(* CODESYS project Cipher-Bay_RECOVERED_2026-03-25T10-42-59.project

Project tree, tasks and I/O mapping:
  Device : CODESYS Control for Linux SL, CODESYS, order no. 2302000005, version 4.19.0.0
    application Application
      libraries: Standard, 3.5.18.0 (System); CmpBitmapPool, * (System)
      task VISU_TASK (cyclic, interval 100 ms, priority 31) calls VisuElems.Visu_Prg
      task MainTask (cyclic, interval t#20ms, priority 1) calls PLC_PRG
      Visualization/
        visualisation VIS_Monitoring
        visualisation VIS_Home
        visualisation VIS_ControlPanel
      POUs/
        program PLC_PRG [ST]
      GLVs/
        global variables GVL_DroneDock
      DUTs/
        data type E_DockState
      External/
        image pool ImagePool
    Ethernet : Ethernet, CODESYS, version 4.2.0.0
        settings: IPAddress = [192,168,0,1]; SubnetMask = [255,255,255,0]; GatewayAddress = [0,0,0,0]; MACAddress = [16#00,16#00,16#00,16#00,16#00,16#00]; NetworkInterfaceName = 'eth0'; NetworkInterfaceName = "eth0"; SaveCommunicationSettings = FALSE; IPAddress = [192,168,0,2]; SubnetMask = [255,255,255,0]; GatewayAddress = [0,0,0,0]
      ModbusTCP_Server_Device : ModbusTCP Server Device, CODESYS, version 4.5.0.0
          settings: DistinctBitAreas = TRUE; Discrete Inputs Size = 16; StartAdresses.DiscreteInputs = 16
          output Application.GVL_DroneDock.mb_iState : WORD  // Input Registers.Input Registers
          output Application.GVL_DroneDock.mb_iBatteryLevel : WORD  // Input Registers.Input Registers
          output Application.GVL_DroneDock.mb_iChargeCurrent : WORD  // Input Registers.Input Registers
          output Application.GVL_DroneDock.xIsDocked : BOOL  // Discrete Inputs.Discrete Inputs.Bit0
          output Application.GVL_DroneDock.xIsCharging : BOOL  // Discrete Inputs.Discrete Inputs.Bit1
          unmapped channels: Holding Registers, Input Registers, Discrete Inputs
    SoftMotion General Axis Pool
  libraries: VisuSymbols, 4.5.0.0 (System); WagoVisuIcons, 1.1.0.9 (WAGO); WagoVisuIconsMaterialDesign, 1.0.0.2 (WAGO)
  text list GlobalTextList
*)

// Device/Application/DUTs/E_DockState
{attribute 'qualified_only'}
{attribute 'strict'}
TYPE E_DockState :
(
	CLOSED := 0,
    OPENING := 1,
    OPEN := 2,
    CLOSING := 3
);
END_TYPE

// Device/Application/GLVs/GVL_DroneDock
VAR_GLOBAL CONSTANT
    // Best Practice: No Magic Numbers
    MAX_BATTERY_LEVEL    : REAL := 100.0;
    CHARGE_CURRENT_MAX   : REAL := 5.2;   // Amps
    CHARGE_RATE_SIM      : REAL := 0.5;   // % added per tick for simulation
    DOOR_TRANSITION_TIME : TIME := T#4S;  // Time it takes to open/close
END_VAR

VAR_GLOBAL
    // HMI Inputs (WebVisu)
    xCmdOpen             : BOOL;
    xCmdClose            : BOOL;
    xCmdSimulateDocking  : BOOL; // Toggle to simulate drone landing

    // System Status
    eCurrentState        : E_DockState := E_DockState.CLOSED;
    xIsDocked            : BOOL;
    xIsCharging          : BOOL;
    rBatteryLevel        : REAL := 20.0; // Start at 20%
    rChargeCurrent       : REAL;

    // Modbus Variables (Scaled for 16-bit Holding Registers)
    // Modbus doesn't handle REALs natively well, so we scale REAL * 10 into INTs
    mb_iState            : WORD;  
	mb_iBatteryLevel     : WORD;  
	mb_iChargeCurrent    : WORD;
    mb_xIsDocked         : BOOL; // Coil
    mb_xIsCharging       : BOOL; // Coil
END_VAR

// Device/Application/POUs/PLC_PRG
PROGRAM PLC_PRG
VAR
	tonDoorTimer   : TON;   // Timer for door opening/closing
    tonChargePulse : TON;   // Timer to pulse the charging simulation
END_VAR

// ==========================================
// 1. DOOR CONTROL STATE MACHINE
// ==========================================
tonDoorTimer(PT := GVL_DroneDock.DOOR_TRANSITION_TIME);

CASE GVL_DroneDock.eCurrentState OF
    
    E_DockState.CLOSED:
        tonDoorTimer(IN := FALSE);
        IF GVL_DroneDock.xCmdOpen THEN
            GVL_DroneDock.xCmdOpen := FALSE; // Consume command
            GVL_DroneDock.eCurrentState := E_DockState.OPENING;
        END_IF

    E_DockState.OPENING:
        tonDoorTimer(IN := TRUE);
        IF tonDoorTimer.Q THEN
            GVL_DroneDock.eCurrentState := E_DockState.OPEN;
        END_IF
        
    E_DockState.OPEN:
        tonDoorTimer(IN := FALSE);
        IF GVL_DroneDock.xCmdClose THEN
            GVL_DroneDock.xCmdClose := FALSE; // Consume command
            GVL_DroneDock.eCurrentState := E_DockState.CLOSING;
        END_IF
        
    E_DockState.CLOSING:
        tonDoorTimer(IN := TRUE);
        IF tonDoorTimer.Q THEN
            GVL_DroneDock.eCurrentState := E_DockState.CLOSED;
        END_IF
        
END_CASE

// ==========================================
// 2. DOCKING & CHARGING SIMULATION LOGIC
// ==========================================
// Drone can only be docked/undocked if the doors are OPEN
IF GVL_DroneDock.eCurrentState = E_DockState.OPEN THEN
    GVL_DroneDock.xIsDocked := GVL_DroneDock.xCmdSimulateDocking;
END_IF

// Charging Logic: Must be docked and doors CLOSED (safe to charge)
IF GVL_DroneDock.xIsDocked AND (GVL_DroneDock.eCurrentState = E_DockState.CLOSED) THEN
    
    IF GVL_DroneDock.rBatteryLevel < GVL_DroneDock.MAX_BATTERY_LEVEL THEN
        GVL_DroneDock.xIsCharging := TRUE;
        GVL_DroneDock.rChargeCurrent := GVL_DroneDock.CHARGE_CURRENT_MAX;
        
        // Simulation: Increase battery level every 1 second
        tonChargePulse(IN := NOT tonChargePulse.Q, PT := T#1S);
        IF tonChargePulse.Q THEN
            GVL_DroneDock.rBatteryLevel := GVL_DroneDock.rBatteryLevel + GVL_DroneDock.CHARGE_RATE_SIM;
        END_IF
    ELSE
        // Battery Full
        GVL_DroneDock.xIsCharging := FALSE;
        GVL_DroneDock.rChargeCurrent := 0.0;
        GVL_DroneDock.rBatteryLevel := GVL_DroneDock.MAX_BATTERY_LEVEL;
    END_IF
    
ELSE
    // Not docked or doors open
    GVL_DroneDock.xIsCharging := FALSE;
    GVL_DroneDock.rChargeCurrent := 0.0;
    tonChargePulse(IN := FALSE);
END_IF

// ==========================================
// 3. MODBUS DATA PREPARATION
// ==========================================
// Convert Enums and REALs into standard WORDs for Modbus transmission
GVL_DroneDock.mb_iState         := INT_TO_WORD(GVL_DroneDock.eCurrentState);
GVL_DroneDock.mb_iBatteryLevel  := REAL_TO_WORD(GVL_DroneDock.rBatteryLevel * 10.0);
GVL_DroneDock.mb_iChargeCurrent := REAL_TO_WORD(GVL_DroneDock.rChargeCurrent * 10.0);
GVL_DroneDock.mb_xIsDocked      := GVL_DroneDock.xIsDocked;
GVL_DroneDock.mb_xIsCharging    := GVL_DroneDock.xIsCharging;

END_PROGRAM

// Device/Application/Visualization/VIS_Monitoring
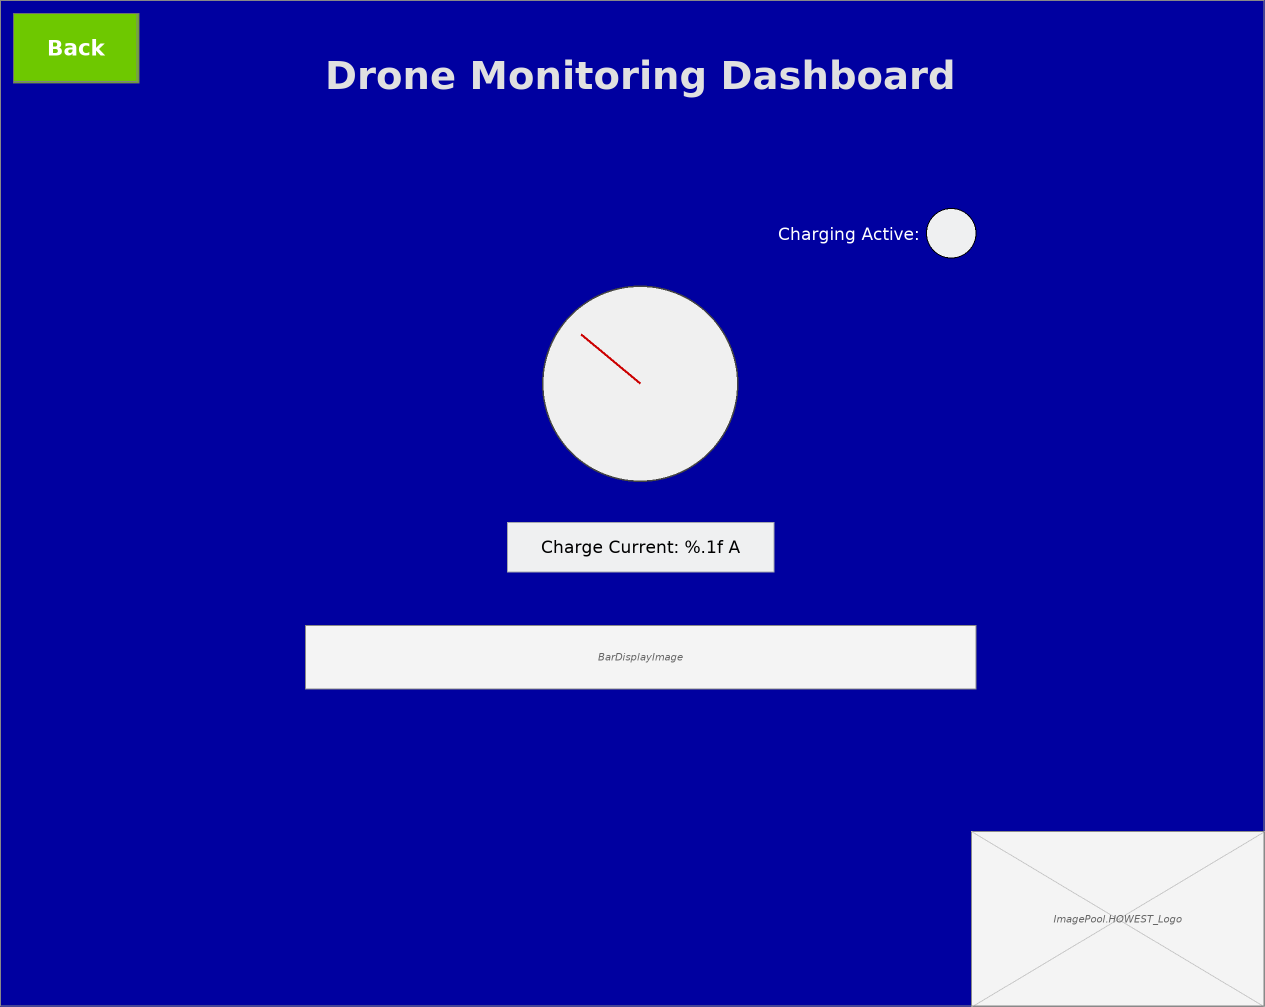
VISUALIZATION VIS_Monitoring  // 1265x1007
    Button (13,13 126x70), "Back"
        OnMouseClick:  Assign=VIS_Home, Type=Assignment
    Label (305,32 671x87), "Drone Monitoring Dashboard"
    BarDisplayImage (305,625 671x64), value: rBatteryLevel, style: BarDisplayImage-Green, scale format: %.1f, scale 0..100
    Rectangle (507,522 267x50), "Charge Current: %.1f A", text variable: rChargeCurrent
    Group (774,208 202x50)
        Ellipse (152,0 50x50), colour toggle: xIsCharging
        Label (0,11 150x30), "Charging Active:"
    Meter360 (542,281 196x205), value: rChargeCurrent, style: Meter-Meter360-Green, scale format: %.1f, scale 0..20
    Image (971,831 294x176), image: ImagePool.HOWEST_Logo
END_VISUALIZATION

// Device/Application/Visualization/VIS_Home
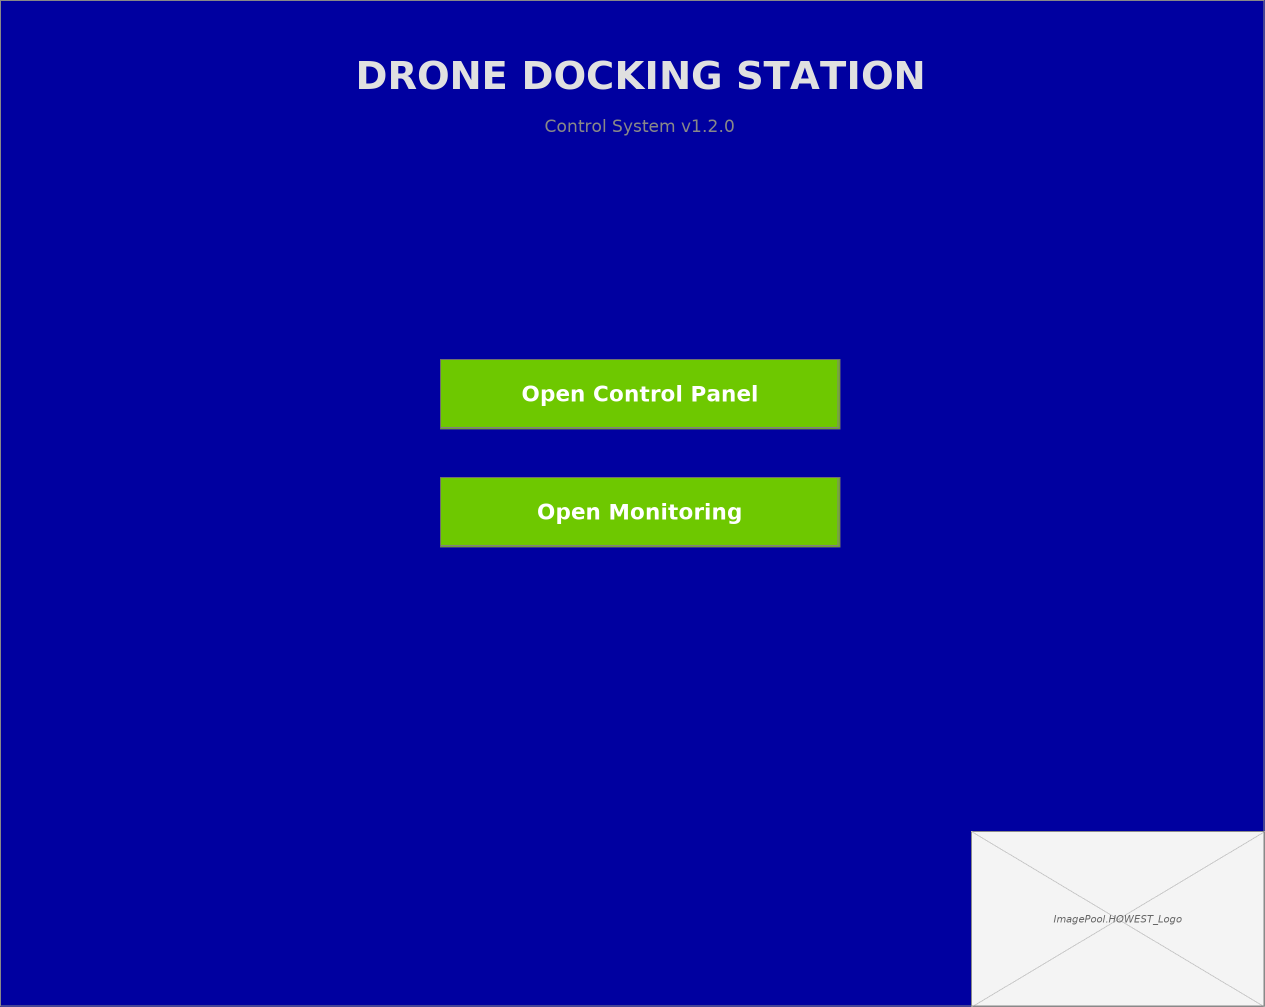
VISUALIZATION VIS_Home  // 1265x1007
    Label (305,32 671x87), "DRONE DOCKING STATION"
    Label (514,109 252x34), "Control System v1.2.0"
    Button (440,359 400x70), "Open Control Panel"
        OnMouseClick:  Assign=VIS_ControlPanel, Type=Assignment
    Button (440,477 400x70), "Open Monitoring"
        OnMouseClick:  Assign=VIS_Monitoring, Type=Assignment
    Image (971,831 294x176), image: ImagePool.HOWEST_Logo
END_VISUALIZATION

// Device/Application/Visualization/VIS_ControlPanel
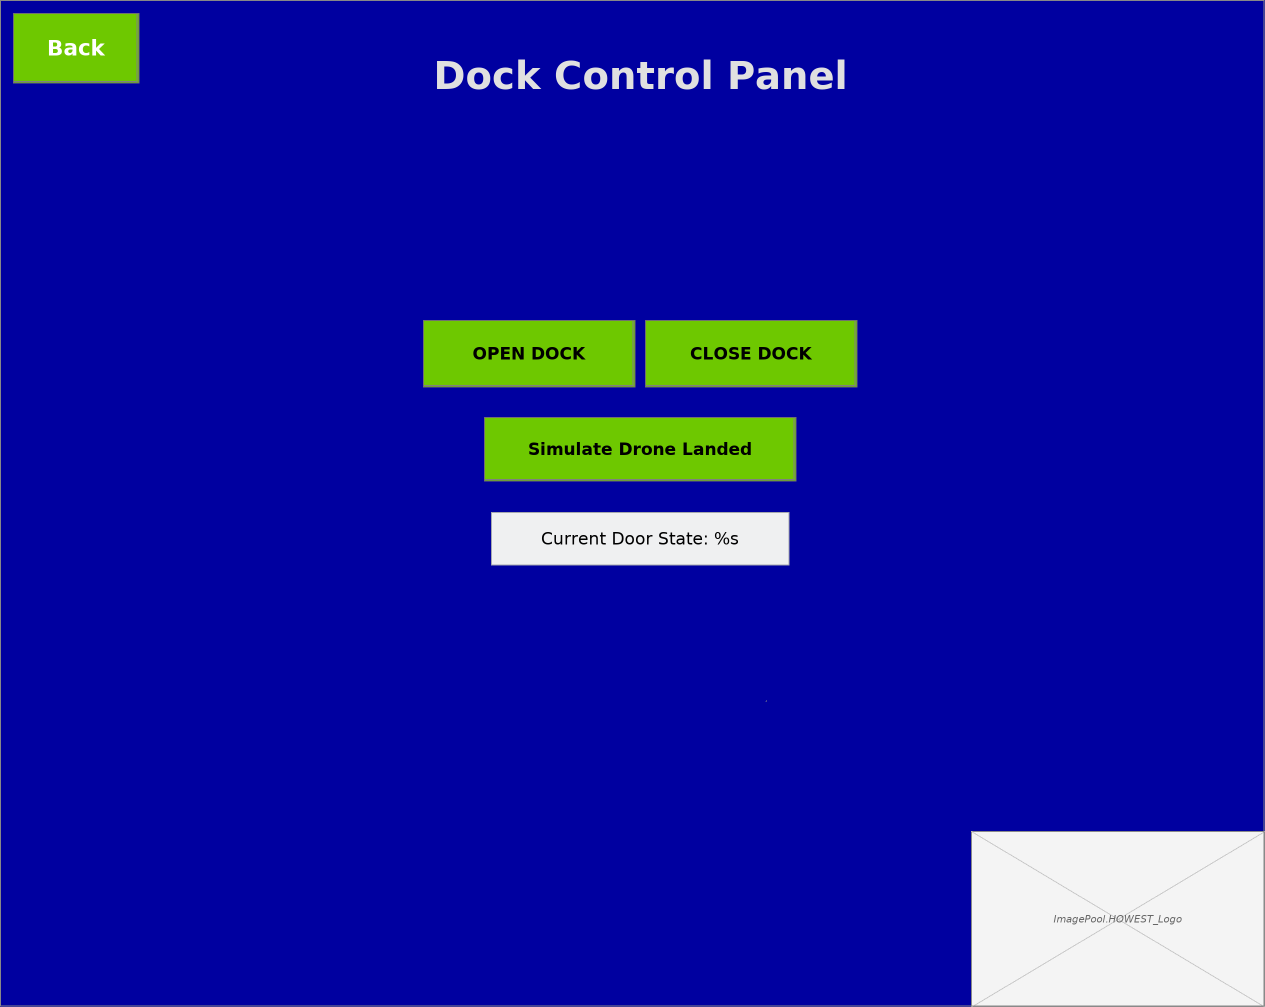
VISUALIZATION VIS_ControlPanel  // 1265x1007
    Button (13,13 126x70), "Back"
        OnMouseClick:  Assign=VIS_Home, Type=Assignment
    Label (305,32 671x87), "Dock Control Panel"
    Button (423,320 212x67), "OPEN DOCK"
        tap xCmdOpen
    Button (645,320 212x67), "CLOSE DOCK"
        tap xCmdClose
    Rectangle (491,512 298x53), "Current Door State: %s", text variable: eCurrentState
    Button (484,417 312x64), "Simulate Drone Landed"
        toggle xCmdSimulateDocking
    WaitingSymbolFlower (766,700 0x1)
    Image (971,831 294x176), image: ImagePool.HOWEST_Logo
END_VISUALIZATION
